(* IEC 61131-3 sources: COTS_ICS_Security/Virtual_Testbed/Workstation/PLC/Editor/build, 2 files *)

(* ---- plc.st ---- *)
TYPE
  LOGLEVEL : (CRITICAL, WARNING, INFO, DEBUG) := INFO;
END_TYPE

FUNCTION_BLOCK LOGGER
  VAR_INPUT
    TRIG : BOOL;
    MSG : STRING;
    LEVEL : LOGLEVEL := INFO;
  END_VAR
  VAR
    TRIG0 : BOOL;
  END_VAR

  IF TRIG AND NOT TRIG0 THEN
  {{
   LogMessage(GetFbVar(LEVEL),(char*)GetFbVar(MSG, .body),GetFbVar(MSG, .len));
  }}
  END_IF;
  TRIG0:=TRIG;
END_FUNCTION_BLOCK

FUNCTION_BLOCK python_eval
  VAR_INPUT
    TRIG : BOOL;
    CODE : STRING;
  END_VAR
  VAR_OUTPUT
    ACK : BOOL;
    RESULT : STRING;
  END_VAR
  VAR
    STATE : DWORD;
    BUFFER : STRING;
    PREBUFFER : STRING;
    TRIGM1 : BOOL;
    TRIGGED : BOOL;
  END_VAR

  {extern void __PythonEvalFB(int, PYTHON_EVAL*);__PythonEvalFB(0, data__);}
END_FUNCTION_BLOCK

FUNCTION_BLOCK python_poll
  VAR_INPUT
    TRIG : BOOL;
    CODE : STRING;
  END_VAR
  VAR_OUTPUT
    ACK : BOOL;
    RESULT : STRING;
  END_VAR
  VAR
    STATE : DWORD;
    BUFFER : STRING;
    PREBUFFER : STRING;
    TRIGM1 : BOOL;
    TRIGGED : BOOL;
  END_VAR

  {extern void __PythonEvalFB(int, PYTHON_EVAL*);__PythonEvalFB(1,(PYTHON_EVAL*)(void*)data__);}
END_FUNCTION_BLOCK

FUNCTION_BLOCK python_gear
  VAR_INPUT
    N : UINT;
    TRIG : BOOL;
    CODE : STRING;
  END_VAR
  VAR_OUTPUT
    ACK : BOOL;
    RESULT : STRING;
  END_VAR
  VAR
    py_eval : python_eval;
    COUNTER : UINT;
    _TMP_ADD10_OUT : UINT;
    _TMP_EQ13_OUT : BOOL;
    _TMP_SEL15_OUT : UINT;
    _TMP_AND7_OUT : BOOL;
  END_VAR

  _TMP_ADD10_OUT := ADD(COUNTER, 1);
  _TMP_EQ13_OUT := EQ(N, _TMP_ADD10_OUT);
  _TMP_SEL15_OUT := SEL(_TMP_EQ13_OUT, _TMP_ADD10_OUT, 0);
  COUNTER := _TMP_SEL15_OUT;
  _TMP_AND7_OUT := AND(_TMP_EQ13_OUT, TRIG);
  py_eval(TRIG := _TMP_AND7_OUT, CODE := CODE);
  ACK := py_eval.ACK;
  RESULT := py_eval.RESULT;
END_FUNCTION_BLOCK

PROGRAM water_tank
  VAR
    Valve_In : BOOL;
    Valve_Out : BOOL;
    Start : BOOL;
    Stop : BOOL;
    High : BOOL;
    Low : BOOL;
    Master : BOOL;
    Height_In : UINT;
    Height_Out : UINT;
    High_Limit : UINT;
    Low_Limit : UINT;
  END_VAR
  VAR
    _TMP_GE19_ENO : BOOL;
    _TMP_GE19_OUT : BOOL;
    _TMP_GT35_ENO : BOOL;
    _TMP_GT35_OUT : BOOL;
    _TMP_MOVE32_ENO : BOOL;
    _TMP_MOVE32_OUT : UINT;
  END_VAR

  Master := NOT(Stop) AND (Master OR Start);
  _TMP_GE19_OUT := GE(EN := Master, IN1 := Height_In, IN2 := High_Limit, ENO => _TMP_GE19_ENO);
  IF _TMP_GE19_ENO THEN
      High := _TMP_GE19_OUT;
  END_IF;
  _TMP_GT35_OUT := GT(EN := Master, IN1 := Height_In, IN2 := Low_Limit, ENO => _TMP_GT35_ENO);
  IF _TMP_GT35_ENO THEN
      Low := _TMP_GT35_OUT;
  END_IF;
  Valve_Out := Low AND (High OR Valve_Out) AND Master;
  Valve_In := NOT(High) AND (NOT(Low) OR NOT(Valve_Out) OR Valve_In) AND Master;
  _TMP_MOVE32_OUT := MOVE(EN := TRUE, IN := Height_In, ENO => _TMP_MOVE32_ENO);
  IF _TMP_MOVE32_ENO THEN
      Height_Out := _TMP_MOVE32_OUT;
  END_IF;
END_PROGRAM

CONFIGURATION Config0

  RESOURCE Res0 ON PLC
    TASK task0(INTERVAL := T#20ms,PRIORITY := 0);
    PROGRAM instance0 WITH task0 : water_tank;
  END_RESOURCE
END_CONFIGURATION

(* ---- generated_plc.st ---- *)
PROGRAM water_tank
  VAR
    Valve_In AT %QX0.0 : BOOL;
    Valve_Out AT %QX0.1 : BOOL;
    Start AT %QX0.2 : BOOL;
    Stop AT %QX0.3 : BOOL;
    High AT %IX0.0 : BOOL;
    Low AT %IX0.1 : BOOL;
    Master AT %IX0.2 : BOOL;
    Height_In AT %IW0 : UINT;
    Height_Out AT %QW0 : UINT;
    High_Limit AT %QW1 : UINT;
    Low_Limit AT %QW2 : UINT;
  END_VAR
  VAR
    _TMP_GE19_ENO : BOOL;
    _TMP_GE19_OUT : BOOL;
    _TMP_GT35_ENO : BOOL;
    _TMP_GT35_OUT : BOOL;
    _TMP_MOVE32_ENO : BOOL;
    _TMP_MOVE32_OUT : UINT;
  END_VAR

  Master := NOT(Stop) AND (Master OR Start);
  _TMP_GE19_OUT := GE(EN := Master, IN1 := Height_In, IN2 := High_Limit, ENO => _TMP_GE19_ENO);
  IF _TMP_GE19_ENO THEN
      High := _TMP_GE19_OUT;
  END_IF;
  _TMP_GT35_OUT := GT(EN := Master, IN1 := Height_In, IN2 := Low_Limit, ENO => _TMP_GT35_ENO);
  IF _TMP_GT35_ENO THEN
      Low := _TMP_GT35_OUT;
  END_IF;
  Valve_Out := Low AND (High OR Valve_Out) AND Master;
  Valve_In := NOT(High) AND (NOT(Low) OR NOT(Valve_Out) OR Valve_In) AND Master;
  _TMP_MOVE32_OUT := MOVE(EN := TRUE, IN := Height_In, ENO => _TMP_MOVE32_ENO);
  IF _TMP_MOVE32_ENO THEN
      Height_Out := _TMP_MOVE32_OUT;
  END_IF;
END_PROGRAM

CONFIGURATION Config0

  RESOURCE Res0 ON PLC
    TASK task0(INTERVAL := T#20ms,PRIORITY := 0);
    PROGRAM instance0 WITH task0 : water_tank;
  END_RESOURCE
END_CONFIGURATION
